// TIA Portal V21 export
TYPE "LBC_typeDigitalSignalProcessValues"
TITLE = LBC_typeDigitalSignalProcessValues
// Module related monitoring information
   STRUCT
      enable { ExternalWritable := 'False'} : Bool;   // Enable functionality of FB
      referenceDesignator { ExternalWritable := 'False'} : WString[154];   // Reference Designator for the module incl. its parent
      simulation { ExternalWritable := 'False'} : Bool;   // Enable simulation input of digital value
      processValue { ExternalWritable := 'False'} : Bool;   // Processed sensor value
      error { ExternalWritable := 'False'} : Bool;   // An error occurred while processing the FB
      status { ExternalWritable := 'False'} : Word;   // 16#0000-16#7FFF: Status of the FB 16#8000-16#FFFF: Error identification
   END_STRUCT;
END_TYPE
